(* Schneider Machine Expert - Basic project Pump_Tank_Backup_System, file version 3.0.0.0 *)

HARDWARE
  EthernetConfiguration: SubnetMask=255.255.255.0
  SerialLineConfiguration: Parity=Even, DataBits=8, StopBits=1

SYMBOLS  (address, symbol, comment, settings)
  %TM0      PUMP1_START_DELAY  "Pump 1 Startup Delay - 2 seconds before speed check"  [Type=TON, TimeBase=TimeBase1s, Preset=2]
  %TM1      PUMP2_START_DELAY  "Pump 2 Startup Delay - 2 seconds before speed check"  [Type=TON, TimeBase=TimeBase1s, Preset=2]
  %TM2      PUMP3_START_DELAY  "Pump 3 Startup Delay - 2 seconds before speed check"  [Type=TON, TimeBase=TimeBase1s, Preset=2]
  %I0.0     START_BTN  "System Start Button"
  %I0.1     STOP_BTN  "System Stop Button (NC)"
  %I0.2     E_STOP  "Emergency Stop (NC)"
  %I0.3     PUMP1_SPEED_OK  "Pump 1 Zero Speed Sensor (NC)"
  %I0.4     PUMP2_SPEED_OK  "Pump 2 Zero Speed Sensor (NC)"
  %I0.5     PUMP3_SPEED_OK  "Pump 3 Zero Speed Sensor (NC)"
  %I0.6     TANK1_LOW  "Tank 1 Low Level Switch"
  %I0.7     TANK1_HIGH  "Tank 1 High Level Switch"
  %I0.8     TANK2_LOW  "Tank 2 Low Level Switch"
  %I0.9     TANK2_HIGH  "Tank 2 High Level Switch"
  %I0.10    TANK3_LOW  "Tank 3 Low Level Switch"
  %I0.11    TANK3_HIGH  "Tank 3 High Level Switch"
  %I0.12    PUMP1_OL  "Pump 1 Overload (NC)"
  %I0.13    PUMP2_OL  "Pump 2 Overload (NC)"
  %I0.14    PUMP3_OL  "Pump 3 Overload (NC)"
  %I0.15    FAULT_RESET  "Fault Reset Button"
  %Q0.0     PUMP1_RUN  "Pump 1 Motor Contactor"
  %Q0.1     PUMP2_RUN  "Pump 2 Motor Contactor"
  %Q0.2     PUMP3_RUN  "Pump 3 Motor Contactor"
  %Q0.3     VALVE_12  "Valve Between Tank 1-2"
  %Q0.4     VALVE_23  "Valve Between Tank 2-3"
  %Q0.5     VALVE_13  "Valve Between Tank 1-3"
  %Q0.6     PUMP1_FAULT_IND  "Pump 1 Fault Indicator"
  %Q0.7     PUMP2_FAULT_IND  "Pump 2 Fault Indicator"
  %Q0.8     PUMP3_FAULT_IND  "Pump 3 Fault Indicator"
  %Q0.9     SYSTEM_RUN_IND  "System Running Indicator"
  %Q0.10    ALARM_OUTPUT  "General Alarm Horn"
  %M0       SYSTEM_RUN  "System Running Flag"
  %M1       PUMP1_CMD  "Pump 1 Command"
  %M2       PUMP2_CMD  "Pump 2 Command"
  %M3       PUMP3_CMD  "Pump 3 Command"
  %M10      PUMP1_FAULT  "Pump 1 Fault (Latched)"
  %M11      PUMP2_FAULT  "Pump 2 Fault (Latched)"
  %M12      PUMP3_FAULT  "Pump 3 Fault (Latched)"
  %M20      TANK1_NEEDS_BACKUP  "Tank 1 Backup Mode"
  %M21      TANK2_NEEDS_BACKUP  "Tank 2 Backup Mode"
  %M22      TANK3_NEEDS_BACKUP  "Tank 3 Backup Mode"

PouDescriptor Pump_Tank_Backup_Main
  (* PouType=Program *)

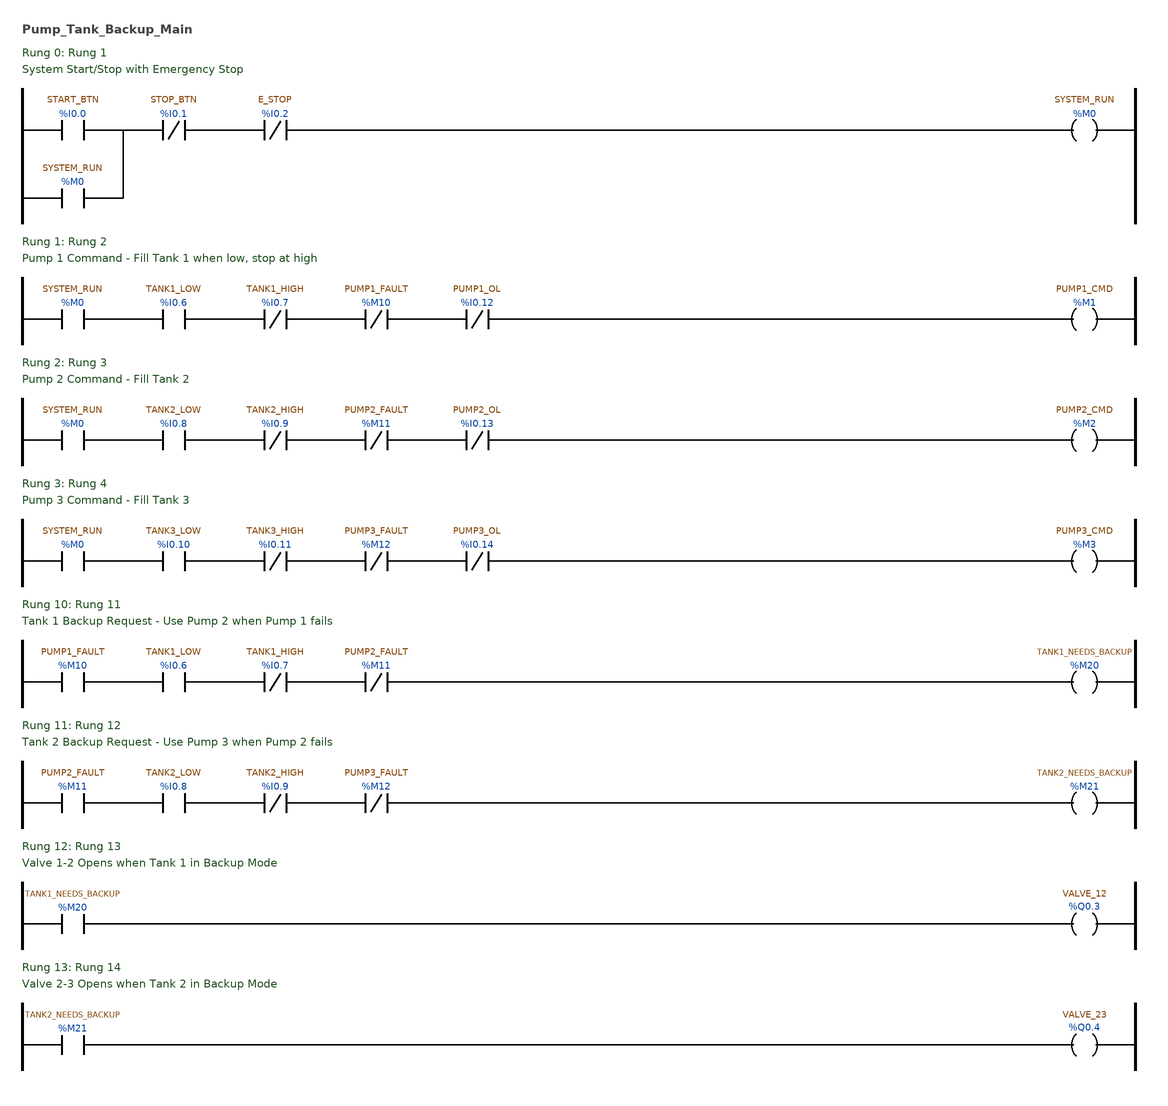

// Rung 0: Rung 1
// System Start/Stop with Emergency Stop
  LD %I0.0                (* START_BTN - Load START button *)
  OR %M0                  (* SYSTEM_RUN - OR with system run flag (seal-in) *)
  ANDN %I0.1              (* STOP_BTN - AND NOT STOP button *)
  ANDN %I0.2              (* E_STOP - AND NOT E-STOP *)
  ST %M0                  (* SYSTEM_RUN - Store to SYSTEM_RUN *)
  // %M0: System Running Seal-in
  // %I0.1: Stop Button (NC)
  // as ST:
  //   SYSTEM_RUN := (START_BTN OR SYSTEM_RUN) AND NOT STOP_BTN AND NOT E_STOP;

// Rung 1: Rung 2
// Pump 1 Command - Fill Tank 1 when low, stop at high
  LD %M0                  (* SYSTEM_RUN - System running *)
  AND %I0.6               (* TANK1_LOW - Tank 1 low level *)
  ANDN %I0.7              (* TANK1_HIGH - Not high level *)
  ANDN %M10               (* PUMP1_FAULT - No pump fault *)
  ANDN %I0.12             (* PUMP1_OL - No overload *)
  ST %M1                  (* PUMP1_CMD - Pump 1 command *)
  // %M0: System Running
  // %I0.6: Tank 1 Low Level
  // %I0.7: Tank 1 High Level (NC)
  // %M10: No Pump 1 Fault
  // %I0.12: No Overload (NC)
  // as ST:
  //   PUMP1_CMD := SYSTEM_RUN AND TANK1_LOW AND NOT TANK1_HIGH AND NOT PUMP1_FAULT AND NOT PUMP1_OL;

// Rung 2: Rung 3
// Pump 2 Command - Fill Tank 2
  LD %M0                  (* SYSTEM_RUN *)
  AND %I0.8               (* TANK2_LOW *)
  ANDN %I0.9              (* TANK2_HIGH *)
  ANDN %M11               (* PUMP2_FAULT *)
  ANDN %I0.13             (* PUMP2_OL *)
  ST %M2                  (* PUMP2_CMD *)
  // %M0: System Running
  // %I0.8: Tank 2 Low Level
  // %I0.9: Tank 2 High Level (NC)
  // %M11: No Pump 2 Fault
  // %I0.13: No Overload (NC)
  // as ST:
  //   PUMP2_CMD := SYSTEM_RUN AND TANK2_LOW AND NOT TANK2_HIGH AND NOT PUMP2_FAULT AND NOT PUMP2_OL;

// Rung 3: Rung 4
// Pump 3 Command - Fill Tank 3
  LD %M0                  (* SYSTEM_RUN *)
  AND %I0.10              (* TANK3_LOW *)
  ANDN %I0.11             (* TANK3_HIGH *)
  ANDN %M12               (* PUMP3_FAULT *)
  ANDN %I0.14             (* PUMP3_OL *)
  ST %M3                  (* PUMP3_CMD *)
  // %M0: System Running
  // %I0.10: Tank 3 Low Level
  // %I0.11: Tank 3 High Level (NC)
  // %M12: No Pump 3 Fault
  // %I0.14: No Overload (NC)
  // as ST:
  //   PUMP3_CMD := SYSTEM_RUN AND TANK3_LOW AND NOT TANK3_HIGH AND NOT PUMP3_FAULT AND NOT PUMP3_OL;

// Rung 4: Rung 5
// Pump 1 Output with Startup Delay Timer
  BLK %TM0                (* PUMP1_START_DELAY - Begin Timer block *)
  LD %M1                  (* PUMP1_CMD - Pump 1 command *)
  IN                      (* Timer input *)
  END_BLK
  LD %M1                  (* PUMP1_CMD *)
  ST %Q0.0                (* PUMP1_RUN - Pump 1 output *)
  // %M1: Pump 1 Command Active
  // %TM0: 2 Second Startup Delay
  // %Q0.0: Pump 1 Motor Output
  // as ST:
  //   PUMP1_START_DELAY(IN := PUMP1_CMD);
  //   PUMP1_RUN := PUMP1_CMD;
  (* the ladder stored for this rung does not match its IL; not drawn *)

// Rung 5: Rung 6
// Pump 1 Zero Speed Fault Detection - Latching
  LD %TM0.Q               (* PUMP1_START_DELAY - Startup delay done *)
  ANDN %I0.3              (* PUMP1_SPEED_OK - Speed not OK *)
  OR %M10                 (* PUMP1_FAULT - OR with fault latch *)
  ANDN %I0.15             (* FAULT_RESET - Not reset *)
  ST %M10                 (* PUMP1_FAULT - Latch fault *)
  // %TM0.Q: Startup Delay Done
  // %M10: Fault Seal-in
  // %I0.3: Speed NOT OK (zero speed)
  // %I0.15: Fault Not Reset
  // %M10: Pump 1 Fault Latched
  // as ST:
  //   PUMP1_FAULT := (PUMP1_START_DELAY.Q AND NOT PUMP1_SPEED_OK OR PUMP1_FAULT) AND NOT FAULT_RESET;
  (* the ladder stored for this rung does not match its IL; not drawn *)

// Rung 6: Rung 7
// Pump 2 Output - Normal or Backup for Tank 1
  LD %M2                  (* PUMP2_CMD *)
  OR %M20                 (* TANK1_NEEDS_BACKUP - OR backup mode for Tank 1 *)
  ST %Q0.1                (* PUMP2_RUN *)
  // %M20: Tank 1 Needs Backup
  // %TM1: 2 Second Startup Delay
  // %Q0.1: Pump 2 Motor Output
  // as ST:
  //   PUMP2_RUN := PUMP2_CMD OR TANK1_NEEDS_BACKUP;
  (* the ladder stored for this rung does not match its IL; not drawn *)

// Rung 7: Rung 8
// Pump 2 Zero Speed Fault Detection
  LD %TM1.Q               (* PUMP2_START_DELAY *)
  ANDN %I0.4              (* PUMP2_SPEED_OK *)
  OR %M11                 (* PUMP2_FAULT *)
  ANDN %I0.15             (* FAULT_RESET *)
  ST %M11                 (* PUMP2_FAULT *)
  // %TM1.Q: Startup Delay Done
  // %M11: Fault Seal-in
  // %I0.4: Speed NOT OK
  // %I0.15: Fault Not Reset
  // %M11: Pump 2 Fault Latched
  // as ST:
  //   PUMP2_FAULT := (PUMP2_START_DELAY.Q AND NOT PUMP2_SPEED_OK OR PUMP2_FAULT) AND NOT FAULT_RESET;
  (* the ladder stored for this rung does not match its IL; not drawn *)

// Rung 8: Rung 9
// Pump 3 Output - Normal or Backup for Tank 2
  LD %M3                  (* PUMP3_CMD *)
  OR %M21                 (* TANK2_NEEDS_BACKUP *)
  ST %Q0.2                (* PUMP3_RUN *)
  // %M21: Tank 2 Needs Backup
  // %TM2: 2 Second Startup Delay
  // %Q0.2: Pump 3 Motor Output
  // as ST:
  //   PUMP3_RUN := PUMP3_CMD OR TANK2_NEEDS_BACKUP;
  (* the ladder stored for this rung does not match its IL; not drawn *)

// Rung 9: Rung 10
// Pump 3 Zero Speed Fault Detection
  LD %TM2.Q               (* PUMP3_START_DELAY *)
  ANDN %I0.5              (* PUMP3_SPEED_OK *)
  OR %M12                 (* PUMP3_FAULT *)
  ANDN %I0.15             (* FAULT_RESET *)
  ST %M12                 (* PUMP3_FAULT *)
  // %TM2.Q: Startup Delay Done
  // %M12: Fault Seal-in
  // %I0.5: Speed NOT OK
  // %I0.15: Fault Not Reset
  // %M12: Pump 3 Fault Latched
  // as ST:
  //   PUMP3_FAULT := (PUMP3_START_DELAY.Q AND NOT PUMP3_SPEED_OK OR PUMP3_FAULT) AND NOT FAULT_RESET;
  (* the ladder stored for this rung does not match its IL; not drawn *)

// Rung 10: Rung 11
// Tank 1 Backup Request - Use Pump 2 when Pump 1 fails
  LD %M10                 (* PUMP1_FAULT - Pump 1 fault *)
  AND %I0.6               (* TANK1_LOW - Tank 1 low *)
  ANDN %I0.7              (* TANK1_HIGH - Not high *)
  ANDN %M11               (* PUMP2_FAULT - Pump 2 available *)
  ST %M20                 (* TANK1_NEEDS_BACKUP *)
  // %M10: Pump 1 Fault Active
  // %I0.6: Tank 1 Low Level
  // %I0.7: Tank 1 Not High
  // %M11: Pump 2 Not Faulted
  // %M20: Tank 1 Needs Backup Fill
  // as ST:
  //   TANK1_NEEDS_BACKUP := PUMP1_FAULT AND TANK1_LOW AND NOT TANK1_HIGH AND NOT PUMP2_FAULT;

// Rung 11: Rung 12
// Tank 2 Backup Request - Use Pump 3 when Pump 2 fails
  LD %M11                 (* PUMP2_FAULT *)
  AND %I0.8               (* TANK2_LOW *)
  ANDN %I0.9              (* TANK2_HIGH *)
  ANDN %M12               (* PUMP3_FAULT *)
  ST %M21                 (* TANK2_NEEDS_BACKUP *)
  // %M11: Pump 2 Fault Active
  // %I0.8: Tank 2 Low Level
  // %I0.9: Tank 2 Not High
  // %M12: Pump 3 Not Faulted
  // %M21: Tank 2 Needs Backup Fill
  // as ST:
  //   TANK2_NEEDS_BACKUP := PUMP2_FAULT AND TANK2_LOW AND NOT TANK2_HIGH AND NOT PUMP3_FAULT;

// Rung 12: Rung 13
// Valve 1-2 Opens when Tank 1 in Backup Mode
  LD %M20                 (* TANK1_NEEDS_BACKUP - Tank 1 backup mode *)
  ST %Q0.3                (* VALVE_12 - Open valve 1-2 *)
  // %M20: Tank 1 Needs Backup
  // %Q0.3: Valve Between Tank 1 and 2
  // as ST:
  //   VALVE_12 := TANK1_NEEDS_BACKUP;

// Rung 13: Rung 14
// Valve 2-3 Opens when Tank 2 in Backup Mode
  LD %M21                 (* TANK2_NEEDS_BACKUP *)
  ST %Q0.4                (* VALVE_23 *)
  // %M21: Tank 2 Needs Backup
  // %Q0.4: Valve Between Tank 2 and 3
  // as ST:
  //   VALVE_23 := TANK2_NEEDS_BACKUP;

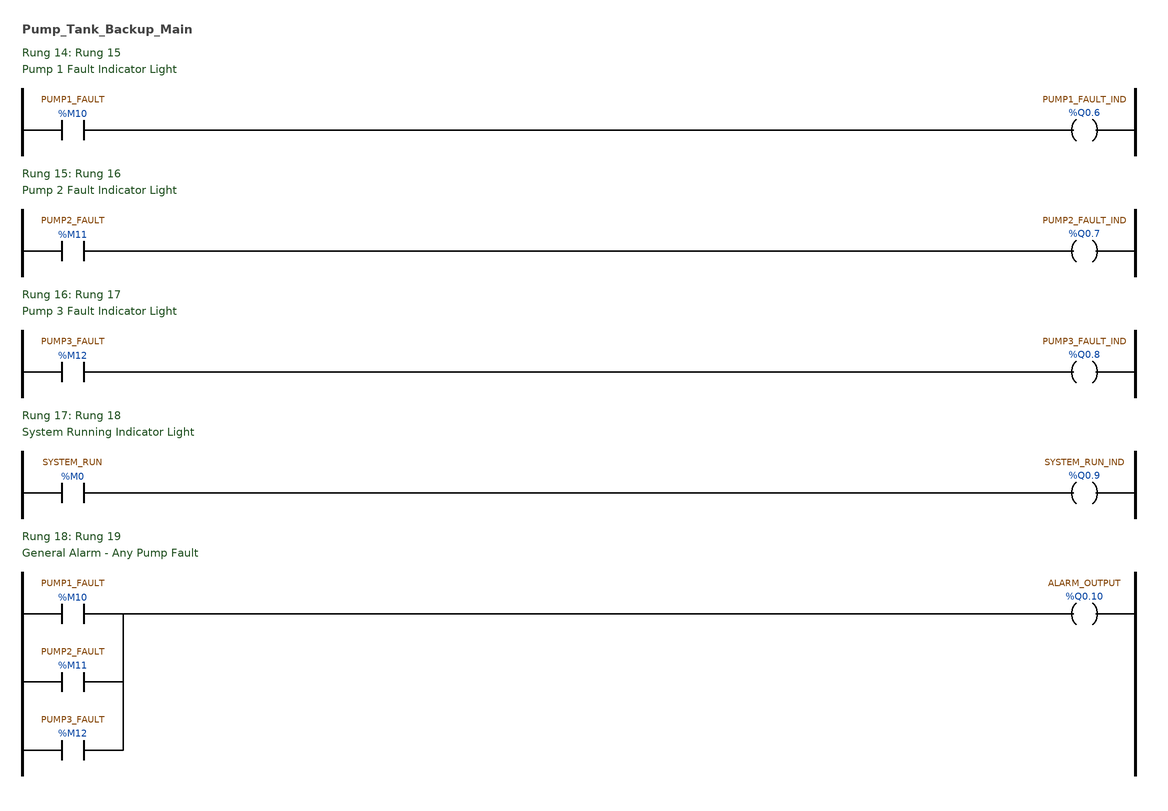

// Rung 14: Rung 15
// Pump 1 Fault Indicator Light
  LD %M10                 (* PUMP1_FAULT *)
  ST %Q0.6                (* PUMP1_FAULT_IND *)
  // %M10: Pump 1 Fault
  // as ST:
  //   PUMP1_FAULT_IND := PUMP1_FAULT;

// Rung 15: Rung 16
// Pump 2 Fault Indicator Light
  LD %M11                 (* PUMP2_FAULT *)
  ST %Q0.7                (* PUMP2_FAULT_IND *)
  // as ST:
  //   PUMP2_FAULT_IND := PUMP2_FAULT;

// Rung 16: Rung 17
// Pump 3 Fault Indicator Light
  LD %M12                 (* PUMP3_FAULT *)
  ST %Q0.8                (* PUMP3_FAULT_IND *)
  // as ST:
  //   PUMP3_FAULT_IND := PUMP3_FAULT;

// Rung 17: Rung 18
// System Running Indicator Light
  LD %M0                  (* SYSTEM_RUN *)
  ST %Q0.9                (* SYSTEM_RUN_IND *)
  // as ST:
  //   SYSTEM_RUN_IND := SYSTEM_RUN;

// Rung 18: Rung 19
// General Alarm - Any Pump Fault
  LD %M10                 (* PUMP1_FAULT *)
  OR %M11                 (* PUMP2_FAULT *)
  OR %M12                 (* PUMP3_FAULT *)
  ST %Q0.10               (* ALARM_OUTPUT *)
  // as ST:
  //   ALARM_OUTPUT := PUMP1_FAULT OR PUMP2_FAULT OR PUMP3_FAULT;
